(* IEC 61131-3 sources: Elmo_Master/Lasal_PRG/Elmo_EtherCAT_Test_4Axis/Class/TCPMotionInterface (part 2) *)

    if (CommandID = 0x7D13) & (Payload = 56) then
      case AxisRef of
        1: controlAxisMask := 0x00000001;
        2: controlAxisMask := 0x00000002;
        3: controlAxisMask := 0x00000004;
        4: controlAxisMask := 0x00000008;
      else
      end_case;
      if (controlAxisMask <> 0) &
         IsClientConnected(#ControlCommands) then
        controlAdmissionResult := ControlCommands.ReserveAxisOwnership(
          CommandId:=0x7D13,
          Reference:=AxisRef$UINT,
          RequestedAxisMask:=controlAxisMask,
          OwnerKind:=3,
          ResourceKind:=2,
          AdmissionMode:=4,
          CallerSessionEpoch:=ActiveRequest.SessionEpoch,
          RequestSequence:=ActiveRequest.Sequence,
          pIdentity:=(#RequestBuf[8])$^void,
          IdentitySize:=Payload$UDINT,
          pEffectiveAxisMask:=#controlEffectiveAxisMask,
          pAdmissionToken:=#controlAdmissionToken,
          pOwnerGeneration:=#controlOwnerGeneration);
        if controlAdmissionResult = 0 then
          controlReserved := TRUE;
        else
          _memset(dest:=#Sendbuf, usByte:=0, cntr:=24);
          Sendbuf[0]$UINT := 0;
          Sendbuf[2]$UINT := 16;
          Sendbuf[4]$UDINT := 0;
          Sendbuf[8]$UINT := 1;
          Sendbuf[10]$UINT := 0;
          Sendbuf[12]$UINT := 1;
          Sendbuf[14]$INT := -31000;
          Sendbuf[16]$UDINT := RequestBuf[12]$UDINT;
          if controlAdmissionResult = -2 then
            Sendbuf[20]$UDINT := 41;
          else
            Sendbuf[20]$UDINT := 42;
          end_if;
          controlResponseSize := 24;
          controlInvokeService := FALSE;
        end_if;
      end_if;
    end_if;

    // LMC_OWNER_ORDINARY_CLASSIFIER_BEGIN
    // Dormant ordinary Axis/Group classifier. The same exact gate is also
    // enforced inside LMCControlCommandService before every native handler.
	  if LMC_AXIS_OWNERSHIP_ORDINARY_ENABLED &
		 (CommandID <> 0x7D13) then
		case CommandID of
        0x2023:
          controlClassifierValid :=
            (Payload = 8) & (AxisRef >= 1) & (AxisRef <= 9) &
            (RequestBuf[8]$UDINT = 1) &
            ((RequestBuf[12] = 0) | (RequestBuf[12] = 1)) &
            (RequestBuf[13] = 1) & (RequestBuf[14] = 0) &
            (RequestBuf[15] = 1);
          controlOwnerKind := LMC_OWNER_KIND_DIRECT;
          controlResourceKind := LMC_OWNER_RESOURCE_AXIS;
          if RequestBuf[12] = 1 then
            controlAdmissionMode := LMC_OWNER_ADMISSION_ORDINARY;
          else
            controlAdmissionMode := LMC_OWNER_ADMISSION_SAFETY;
          end_if;
        0x2024:
          controlClassifierValid :=
            (Payload = 1) & (AxisRef >= 1) & (AxisRef <= 9) &
            (RequestBuf[8] = 1);
          controlOwnerKind := LMC_OWNER_KIND_DIRECT;
          controlResourceKind := LMC_OWNER_RESOURCE_AXIS;
          controlAdmissionMode := LMC_OWNER_ADMISSION_ORDINARY;
        0x2022:
          controlClassifierValid :=
            (Payload = 16) & (AxisRef >= 1) & (AxisRef <= 9) &
            (RequestBuf[8]$DINT > 0) &
            (RequestBuf[12]$DINT >= 0) &
            (RequestBuf[16]$DINT = 1) &
            (RequestBuf[20]$DINT = 1);
          controlOwnerKind := LMC_OWNER_KIND_DIRECT;
          controlResourceKind := LMC_OWNER_RESOURCE_AXIS;
          controlAdmissionMode := LMC_OWNER_ADMISSION_SAFETY;
        0x209F, 0x20A0:
          controlClassifierValid :=
            (Payload = 32) & (AxisRef >= 1) & (AxisRef <= 9) &
            (RequestBuf[28]$DINT = 2) &
            (RequestBuf[32]$DINT = 1) &
            (RequestBuf[36]$DINT = 1);
          controlOwnerKind := LMC_OWNER_KIND_DIRECT;
          controlResourceKind := LMC_OWNER_RESOURCE_AXIS;
          controlAdmissionMode := LMC_OWNER_ADMISSION_ORDINARY;
        0x20A2:
          controlClassifierValid :=
            (Payload = 24) & (AxisRef >= 1) & (AxisRef <= 9) &
            (RequestBuf[16]$DINT = 0) &
            (RequestBuf[28]$DINT = 1) &
            (((RequestBuf[24]$DINT = 1) &
              (RequestBuf[8]$DINT >= 0)) |
             ((RequestBuf[24]$DINT = 3) &
              (RequestBuf[8]$DINT <= 0)));
          controlOwnerKind := LMC_OWNER_KIND_DIRECT;
          controlResourceKind := LMC_OWNER_RESOURCE_AXIS;
          controlAdmissionMode := LMC_OWNER_ADMISSION_ORDINARY;
        0x2047:
          controlClassifierValid :=
            (Payload = 1) & (AxisRef = 0x0100) &
            (RequestBuf[8] = 1);
          controlAxisMask := LMC_OWNER_PROFILE_AXIS_MASK;
          controlOwnerKind := LMC_OWNER_KIND_GROUP;
          controlResourceKind := LMC_OWNER_RESOURCE_AXIS;
          controlAdmissionMode := LMC_OWNER_ADMISSION_ORDINARY;
        0x2048:
          controlClassifierValid :=
            (Payload = 1) & (AxisRef = 0x0100) &
            (RequestBuf[8] = 1);
          controlAxisMask := LMC_OWNER_PROFILE_AXIS_MASK;
          controlOwnerKind := LMC_OWNER_KIND_GROUP;
          controlResourceKind := LMC_OWNER_RESOURCE_AXIS;
          controlAdmissionMode := LMC_OWNER_ADMISSION_SAFETY;
        0x2049, 0x204A:
          controlClassifierValid :=
            (Payload = 1) & (AxisRef = 0x0100) &
            (RequestBuf[8] = 1);
          controlAxisMask := LMC_OWNER_ROBOT_AXIS_MASK;
          controlOwnerKind := LMC_OWNER_KIND_GROUP;
          controlResourceKind := LMC_OWNER_RESOURCE_AXIS;
          controlAdmissionMode := LMC_OWNER_ADMISSION_ORDINARY;
        0x204B:
          controlClassifierValid :=
            (Payload = 1) & (AxisRef = 0x0100) &
            (RequestBuf[8] = 1);
          controlAxisMask := LMC_OWNER_ROBOT_AXIS_MASK;
          controlOwnerKind := LMC_OWNER_KIND_GROUP;
          controlResourceKind := LMC_OWNER_RESOURCE_AXIS;
          controlAdmissionMode := LMC_OWNER_ADMISSION_SAFETY;
        0x2085:
          controlClassifierValid :=
            (Payload = 16) & (AxisRef = 0x0100) &
            (RequestBuf[8]$DINT >= 0) &
            (RequestBuf[12]$DINT >= 0) &
            (RequestBuf[16]$DINT = 1) &
            (RequestBuf[20]$DINT = 1) &
            ((RequestBuf[12]$DINT = 0) |
             (RequestBuf[8]$DINT > 0));
          controlAxisMask := LMC_OWNER_PROFILE_AXIS_MASK;
          controlOwnerKind := LMC_OWNER_KIND_GROUP;
          controlResourceKind := LMC_OWNER_RESOURCE_AXIS;
          controlAdmissionMode := LMC_OWNER_ADMISSION_SAFETY;
        0x20A4:
          controlClassifierValid :=
            (Payload = 96) & (AxisRef = 0x0100) &
            (RequestBuf[72]$DINT > 0) &
            (RequestBuf[76]$DINT > 0) &
            (RequestBuf[80]$DINT > 0) &
            (RequestBuf[84]$DINT >= 0) &
            (RequestBuf[88]$DINT = 0) &
            ((RequestBuf[92]$DINT = 0) |
             (RequestBuf[92]$DINT = 2)) &
            ((RequestBuf[96]$DINT = 1) |
             (RequestBuf[96]$DINT = 2)) &
            (RequestBuf[100]$DINT = 1);
          controlIdentityIndex := 4;
          while controlIdentityIndex <= 15 do
            if RequestBuf[8 + (controlIdentityIndex * 4)]$DINT <> 0 then
              controlClassifierValid := FALSE;
            end_if;
            controlIdentityIndex += 1;
          end_while;
          controlAxisMask := LMC_OWNER_PROFILE_AXIS_MASK;
          controlOwnerKind := LMC_OWNER_KIND_GROUP;
          controlResourceKind := LMC_OWNER_RESOURCE_AXIS;
          controlAdmissionMode := LMC_OWNER_ADMISSION_ORDINARY;
        0x7D22:
          controlClassifierValid :=
            (Payload = 104) & (AxisRef = 0x0100) &
            (RequestBuf[8]$UINT = 1) &
            (RequestBuf[10]$UINT = 0) &
            (RequestBuf[12]$UDINT <> 0) &
            (RequestBuf[80]$DINT > 0) &
            (RequestBuf[84]$DINT > 0) &
            (RequestBuf[88]$DINT > 0) &
            (RequestBuf[92]$DINT >= 0) &
            (RequestBuf[96]$DINT = 0) &
            ((RequestBuf[100]$DINT = 0) |
             (RequestBuf[100]$DINT = 2)) &
            ((RequestBuf[104]$DINT = 1) |
             (RequestBuf[104]$DINT = 2)) &
            (RequestBuf[108]$DINT = 1);
          controlIdentityIndex := 4;
          while controlIdentityIndex <= 15 do
            if RequestBuf[16 + (controlIdentityIndex * 4)]$DINT <> 0 then
              controlClassifierValid := FALSE;
            end_if;
            controlIdentityIndex += 1;
          end_while;
          controlAxisMask := LMC_OWNER_PROFILE_AXIS_MASK;
          controlOwnerKind := LMC_OWNER_KIND_GROUP;
          controlResourceKind := LMC_OWNER_RESOURCE_AXIS;
          controlAdmissionMode := LMC_OWNER_ADMISSION_ORDINARY;
        0x20E7:
          controlClassifierValid :=
            (Payload = 1320) & (AxisRef = 0x0100);
          controlAxisMask := LMC_OWNER_ROBOT_AXIS_MASK;
          controlOwnerKind := LMC_OWNER_KIND_GROUP;
          controlResourceKind := LMC_OWNER_RESOURCE_AXIS;
          controlAdmissionMode := LMC_OWNER_ADMISSION_LIFECYCLE;
      else
      end_case;
		controlManagedCommand := controlOwnerKind <> 0;
		if controlClassifierValid &
		   (controlOwnerKind = LMC_OWNER_KIND_DIRECT) then
        case AxisRef of
          1: controlAxisMask := 0x00000001;
          2: controlAxisMask := 0x00000002;
          3: controlAxisMask := 0x00000004;
          4: controlAxisMask := 0x00000008;
          5: controlAxisMask := 0x00000010;
          6: controlAxisMask := 0x00000020;
          7: controlAxisMask := 0x00000040;
          8: controlAxisMask := 0x00000080;
          9: controlAxisMask := 0x00000100;
        else
          controlAxisMask := 0;
        end_case;
		end_if;
		if controlManagedCommand & (controlClassifierValid = FALSE) then
		  controlInvokeService := FALSE;
		end_if;

		if controlClassifierValid & (controlAxisMask <> 0) then
        if IsClientConnected(#ControlCommands) then
          controlAdmissionResult := ControlCommands.ReserveAxisOwnership(
            CommandId:=CommandID$UINT,
            Reference:=AxisRef$UINT,
            RequestedAxisMask:=controlAxisMask,
            OwnerKind:=controlOwnerKind,
            ResourceKind:=controlResourceKind,
            AdmissionMode:=controlAdmissionMode,
            CallerSessionEpoch:=ActiveRequest.SessionEpoch,
            RequestSequence:=ActiveRequest.Sequence,
            pIdentity:=(#RequestBuf[8])$^void,
            IdentitySize:=Payload$UDINT,
            pEffectiveAxisMask:=#controlEffectiveAxisMask,
            pAdmissionToken:=#controlAdmissionToken,
            pOwnerGeneration:=#controlOwnerGeneration);
        else
          controlAdmissionResult := -3;
        end_if;
		if controlAdmissionResult < 0 then
          if CommandID = 0x7D22 then
            _memset(dest:=#Sendbuf, usByte:=0, cntr:=24);
            Sendbuf[0]$UINT := 0;
            Sendbuf[2]$UINT := 16;
            Sendbuf[8]$UINT := 1;
            Sendbuf[12]$UINT := 1;
            Sendbuf[14]$INT := -31000;
            Sendbuf[16]$UDINT := RequestBuf[12]$UDINT;
            if controlAdmissionResult = -2 then
              Sendbuf[20]$UDINT := 41;
            else
              Sendbuf[20]$UDINT := 42;
            end_if;
            controlResponseSize := 24;
          elsif CommandID = 0x20E7 then
            _memset(dest:=#Sendbuf, usByte:=0, cntr:=12);
            Sendbuf[0]$UINT := 0;
            Sendbuf[2]$UINT := 4;
            Sendbuf[8]$UINT := 1;
            Sendbuf[10]$INT := LMC_OWNER_ADAPTER_ERROR_CONFLICT;
            controlResponseSize := 12;
          else
            _memset(dest:=#Sendbuf, usByte:=0, cntr:=16);
            Sendbuf[0]$UINT := 0;
            Sendbuf[2]$UINT := 8;
            Sendbuf[8]$UDINT := TO_UDINT(AxisRef);
            Sendbuf[12]$UINT := 1;
            Sendbuf[14]$INT := LMC_OWNER_ADAPTER_ERROR_CONFLICT;
            controlResponseSize := 16;
          end_if;
          controlInvokeService := FALSE;
        end_if;
      end_if;
    end_if;
    // LMC_OWNER_ORDINARY_CLASSIFIER_END
	  end_if;

    if controlInvokeService & IsClientConnected(#ControlCommands) then
      controlResponseSize := ControlCommands.HandleRequest(
        CommandId:=CommandID$UINT,
        Reference:=AxisRef$UINT,
        pRequestFrame:=(#RequestBuf[0])$^USINT,
        RequestFrameSize:=(Payload + 8)$UDINT,
        pResponseFrame:=(#Sendbuf[0])$^USINT,
        ResponseCapacity:=sizeof(Sendbuf),
        CallerSessionEpoch:=ActiveRequest.SessionEpoch,
        RequestSequence:=ActiveRequest.Sequence,
        AdmissionToken:=controlAdmissionToken,
        OwnerGeneration:=controlOwnerGeneration,
        ResponseSocket:=ActiveRequest.Socket);
    end_if;

    // LMC_ADMIN_SET_POSITION_PENDING_BEGIN
    if (CommandID = 0x7D12) &
       (controlResponseSize = LMC_ADMIN_SET_POSITION_PENDING) then
      setPositionPendingResult := HandleAdminSetPositionPending(
        Phase:=LMC_ADMIN_SET_POSITION_PENDING_PHASE_RETAIN);
      if setPositionPendingResult = 1 then
        ActiveRequestValid := TRUE;
      end_if;
      RETURN;
    end_if;
    if CommandID = 0x7D12 then
      setPositionPendingResult := HandleAdminSetPositionPending(
        Phase:=LMC_ADMIN_SET_POSITION_PENDING_PHASE_TERMINAL);
    end_if;
    // LMC_ADMIN_SET_POSITION_PENDING_END

    // LMC_ADMIN_SET_POSITION_QUARANTINE_BEGIN
    if (CommandID = 0x7D12) &
       (controlResponseSize =
        LMC_ADMIN_SET_POSITION_QUARANTINE_CLOSE) then
      setPositionPendingResult := HandleAdminSetPositionPending(
        Phase:=LMC_ADMIN_SET_POSITION_PENDING_PHASE_QUARANTINE);
      RETURN;
    end_if;
    // LMC_ADMIN_SET_POSITION_QUARANTINE_END

    // LMC_ADMIN_SET_POSITION_CLOSE_WITHOUT_RESPONSE_BEGIN
    if (CommandID = 0x7D12) &
       (controlResponseSize =
        LMC_ADMIN_SET_POSITION_CLOSE_WITHOUT_RESPONSE) then
      setPositionCloseSocket := ActiveRequest.Socket;
      if (ActiveRequest.SessionEpoch <> 0) &
         (PendingClosedSessionEpoch = 0) then
        PendingClosedSessionEpoch := ActiveRequest.SessionEpoch;
        callbackDisarmResult := DisarmRpcCallbackEndpoint();
        SessionEpoch += 1;
        if SessionEpoch = 0 then
          SessionEpoch := 1;
        end_if;
      end_if;
      IngressBlocked := TRUE;
      IngressFaultPending := FALSE;
      IngressFaultCloseRequired := TRUE;
      RpcSocket := 0;
      RpcInitialized := FALSE;
      if setPositionCloseSocket <> 0 then
        LastOwnerDisconnectRequestRet :=
          _TCPIPServerInterface::SetSocketParameter(
            dSock:=setPositionCloseSocket,
            Cmd:=100,
            SubCmd:=0,
            ParaValue:=0
          );
      end_if;
      RETURN;
    end_if;
    // LMC_ADMIN_SET_POSITION_CLOSE_WITHOUT_RESPONSE_END

    if controlResponseSize = LMC_OWNER_SAFETY_DRAIN_PENDING then
		controlPendingResult := HandleControlSafetyDrainPending(
		  Phase:=LMC_OWNER_SAFETY_PHASE_RETAIN,
		  EffectiveAxisMask:=controlEffectiveAxisMask,
		  AdmissionToken:=controlAdmissionToken,
		  OwnerGeneration:=controlOwnerGeneration);
		RETURN;
	  elsif controlPendingContinuation then
		ActiveRequest.PayloadData[
		  LMC_OWNER_SAFETY_PENDING_RESPONSE_OFFSET]$DINT :=
		  controlResponseSize;
		controlPendingResult := HandleControlSafetyDrainPending(
		  Phase:=LMC_OWNER_SAFETY_PHASE_TERMINAL,
		  EffectiveAxisMask:=controlEffectiveAxisMask,
		  AdmissionToken:=controlAdmissionToken,
		  OwnerGeneration:=controlOwnerGeneration);
		RETURN;
		elsif controlReserved then
      controlExactAccepted :=
        (controlResponseSize = 32) &
        (Sendbuf[0]$UINT = 0) &
        (Sendbuf[2]$UINT = 24) &
        (Sendbuf[8]$UINT = 1) &
        (Sendbuf[12]$UINT = 0) &
        (Sendbuf[14]$INT = 0) &
        (Sendbuf[16]$UDINT = RequestBuf[12]$UDINT) &
        (Sendbuf[24]$UINT = 1) &
        (Sendbuf[26]$UINT = 0) &
        (Sendbuf[28]$UDINT = 0);
      controlExactFailure :=
        (controlResponseSize = 24) &
        (Sendbuf[0]$UINT = 0) &
        (Sendbuf[2]$UINT = 16) &
        (Sendbuf[8]$UINT = 1) &
        (Sendbuf[12]$UINT = 1) &
        (Sendbuf[14]$INT = -31000) &
        (Sendbuf[16]$UDINT = RequestBuf[12]$UDINT) &
        (((Sendbuf[20]$UDINT >= 1) &
          (Sendbuf[20]$UDINT <= 5)) |
         (Sendbuf[20]$UDINT = 10) |
         (Sendbuf[20]$UDINT = 13) |
         ((Sendbuf[20]$UDINT >= 15) &
          (Sendbuf[20]$UDINT <= 18)) |
         ((Sendbuf[20]$UDINT >= 40) &
          (Sendbuf[20]$UDINT <= 42)));
      if (controlExactAccepted = FALSE) &
         (controlExactFailure = FALSE) then
        _memset(dest:=#Sendbuf, usByte:=0, cntr:=24);
        Sendbuf[0]$UINT := 0;
        Sendbuf[2]$UINT := 16;
        Sendbuf[8]$UINT := 1;
        Sendbuf[12]$UINT := 1;
        Sendbuf[14]$INT := -31000;
        Sendbuf[16]$UDINT := RequestBuf[12]$UDINT;
        Sendbuf[20]$UDINT := 42;
        controlResponseSize := 24;
      end_if;
    end_if;

      if (controlResponseSize <= 0) |
         (controlResponseSize > sizeof(Sendbuf)) then
        _memset(dest:=#Sendbuf, usByte:=0, cntr:=sizeof(Sendbuf));
        Sendbuf[0]$UINT := 1;
        Sendbuf[2]$UINT := 4;
        Sendbuf[4]$UDINT := 0;
        Sendbuf[8]$UINT := 1;
        Sendbuf[10]$INT := -1;
        controlResponseSize := 12;
      end_if;

      SendData(
        pData:=#Sendbuf[0],
        udSize:=controlResponseSize$UDINT,
        dSocket:=CurrentSock,
        bDirect:=TRUE
      );

  else
    _memset(dest:=#Sendbuf, usByte:=0, cntr:=sizeof(Sendbuf));
    Sendbuf[0]$UINT := 1;
    Sendbuf[2]$UINT := 4;
    Sendbuf[4]$UDINT := 0;
    Sendbuf[8]$UINT := 1;
    Sendbuf[10]$INT := -4;
    SendData(pData:=#Sendbuf[0], udSize:=12,
             dSocket:=CurrentSock, bDirect:=TRUE);
end_case;

END_FUNCTION

FUNCTION TCPMotionInterface::DisarmRpcCallbackEndpoint
	VAR_OUTPUT
		Result 	: DINT;
	END_VAR

	Result := 1;
	IF (RpcCallbackProtocolVersion <> 2) OR
	   (RpcCallbackRegistered = FALSE) THEN
		Result := 1;
	// IsClientConnected returns an integer; NOT would bitwise-invert it.
	ELSIF IsClientConnected(#CallbackSender) = 0 THEN
		Result := -9;
	ELSE
		Result := CallbackSender.DisarmEndpoint(
			ExpectedSessionEpoch := RpcCallbackSessionEpoch,
			ExpectedCookieLo := RpcCallbackCookieLo,
			ExpectedCookieHi := RpcCallbackCookieHi
		);
	END_IF;
	// A dormant no-op must not overwrite completed owner-loss evidence.
	IF RpcCallbackRegistered THEN
		RpcCallbackLastDisarmResult := Result;
	END_IF;
	IF (Result = 0) OR (Result = 1) THEN
		RpcCallbackRegistered := FALSE;
		RpcCallbackEventMask := 0;
		RpcCallbackPort := 0;
		RpcCallbackIPv4[0] := 0;
		RpcCallbackIPv4[1] := 0;
		RpcCallbackIPv4[2] := 0;
		RpcCallbackIPv4[3] := 0;
		RpcCallbackProtocolVersion := 0;
		RpcCallbackAcceptedMaxDatagram := 0;
		RpcCallbackSessionEpoch := 0;
		RpcCallbackBootId := 0;
		RpcCallbackCookieLo := 0;
		RpcCallbackCookieHi := 0;
	END_IF;
END_FUNCTION

FUNCTION TCPMotionInterface::PublishD5TerminalWake
	VAR
		ticketId : UDINT;
		ticketBootId : UDINT;
		ownerSessionEpoch : UDINT;
		takeResult : DINT;
		publishResult : DINT;
	END_VAR

	ticketId := 0;
	ticketBootId := 0;
	ownerSessionEpoch := 0;
	if IsClientConnected(#Diagnostics) = FALSE then
		RETURN;
	end_if;
	takeResult := Diagnostics.TryTakeD5TerminalWake(
		pTicketId:=#ticketId,
		pTicketBootId:=#ticketBootId,
		pOwnerSessionEpoch:=#ownerSessionEpoch);
	if takeResult <> 1 then
		RETURN;
	end_if;

	if D5TerminalWakeAttemptCount <> 16#FFFFFFFF then
		D5TerminalWakeAttemptCount += 1;
	end_if;
	publishResult := -9;
	if RpcInitialized & (CurrentSock <> 0) & (RpcSocket = CurrentSock) &
		(PendingClosedSessionEpoch = 0) &
		RpcCallbackRegistered & (RpcCallbackProtocolVersion = 2) &
		((RpcCallbackEventMask AND 1) = 1) &
		(RpcCallbackSessionEpoch = SessionEpoch) &
		(ownerSessionEpoch = RpcCallbackSessionEpoch) &
		(ticketBootId = RpcCallbackBootId) &
		IsClientConnected(#CallbackSender) then
		publishResult := CallbackSender.PublishEvent(
			EventMaskBit:=1,
			EventType:=1,
			DeliveryClass:=0,
			EventId:=ticketId,
			ProducerSessionEpoch:=ownerSessionEpoch,
			pPayload:=NIL,
			PayloadBytes:=0);
	end_if;
	if publishResult = 0 then
		if D5TerminalWakeEnqueuedCount <> 16#FFFFFFFF then
			D5TerminalWakeEnqueuedCount += 1;
		end_if;
	else
		if D5TerminalWakeRejectedCount <> 16#FFFFFFFF then
			D5TerminalWakeRejectedCount += 1;
		end_if;
	end_if;

END_FUNCTION
